// TIA Portal V19 export
DATA_BLOCK "ManualOperationControl_Template"   // DB91
// stored: MemoryReserve 100
   VAR
      manualOperationEm { ExternalAccessible := 'False'; ExternalVisible := 'False'; ExternalWritable := 'False'} : "LAF_typeManEm";
      manualOperationEmArea { ExternalAccessible := 'False'; ExternalVisible := 'False'; ExternalWritable := 'False'} : Array[1..1] of "LAF_typeManOperationArea";
      manualOperationCms { ExternalAccessible := 'False'; ExternalVisible := 'False'; ExternalWritable := 'False'} : Array[1..1] of "LAF_typeManOperation";
   END_VAR
BEGIN
   manualOperationEm.equipmentModuleNum := 3400;
END_DATA_BLOCK
